// TwinCAT 3 PLC project Untitled1
// ProgramVersion: 3.1.4023.0
// libraries:
//   CmpBitmapPool, * (System)
//   Tc2_MC2, * (Beckhoff Automation GmbH)
//   Tc2_Standard, * (Beckhoff Automation GmbH)
//   Tc2_System, * (Beckhoff Automation GmbH)
//   Tc2_Utilities, * (Beckhoff Automation GmbH)
//   Tc3_Module, * (Beckhoff Automation GmbH)
//   Tc3_PackML_V2, * (Beckhoff Automation GmbH)
// project tree:
//   DUTs/ A21ToolStorage.TcDUT (not stored), Bundle.TcDUT (not stored), EOAT.TcDUT (not stored), Interval.TcDUT (not stored), PositionMaterials.TcDUT (not stored)
//   DUTs/Enums/ A21.TcDUT (not stored), Chipboard.TcDUT (not stored), Homing.TcDUT (not stored), SectionEnum.TcDUT (not stored), Surface.TcDUT, WoodBunk.TcDUT (not stored)
//   DUTs/Insertion/Drives/ AirPiston.TcPOU (not stored), ClearLinkMC.TcPOU (not stored), SimplePiston.TcPOU (not stored)
//   DUTs/Insertion/ Insertion.TcPOU (not stored), SuctionPad.TcDUT (not stored)
//   DUTs/Insertion/Prototypes/ FBA_Drive.TcPOU (not stored), I_ContinuousDrive.TcIO (not stored), I_Drive.TcIO, I_PositionalDrive.TcIO (not stored), I_EncodedDrive.TcIO (not stored)
//   DUTs/Machines/ Conveyor.TcPOU, ConveyorMode.TcDUT (not stored), KukaRobot.TcPOU (not stored), RobotA21.TcPOU (not stored), StrapMachine.TcPOU (not stored)
//   DUTs/Material Holders/ MaterialHolder.TcPOU (not stored), MaterialSlot.TcDUT (not stored), SkidMagazine.TcPOU (not stored), StagingTable.TcPOU (not stored)
//   GVLs/ ContainerArrays.TcGVL (not stored), GVL.TcGVL (not stored), Hardware.TcGVL (not stored), Misc.TcGVL (not stored)
//   / PlcTask.TcTTO (not stored)
//   POUs/A21a - Chipboard/AOIs/ AOI_LoadChipboard.TcPOU (not stored)
//   POUs/A21b - Wood Bunk/AOIs/ AOI_LoadWoodBunk.TcPOU (not stored), AOI_WoodBunkAlarms.TcPOU (not stored), AOI_StageWoodBunk.TcPOU (not stored), AOI_StagingTemplate.TcPOU (not stored)
//   POUs/ FB_System.TcPOU (not stored), MAIN.TcPOU
//   POUs/Hardware Calls/ InsertionQuality.TcPOU (not stored), SetSuctionsPtrArr.TcPOU (not stored), SuctionQuality.TcPOU (not stored), CallHardware.TcPOU (not stored), SetSuctions.TcPOU (not stored), SetupHardware.TcPOU (not stored)
//   POUs/A21a - Chipboard/ ChipboardEx.TcPOU (not stored)
//   POUs/A21b - Wood Bunk/ WoodBunkEx.TcPOU
//   POUs/Utility/ AddToStringArray.TcPOU (not stored), ArrayIsEmpty.TcPOU (not stored), BoolVLArrayToInteger.TcPOU (not stored), BoolPtrArrayToInteger.TcPOU (not stored), CleanStringsArray.TcPOU (not stored), IntegerBitAccess.TcPOU (not stored), IntegerToBoolArray.TcPOU (not stored), JoinStrings.TcPOU (not stored), WithinTolerance.TcPOU (not stored)

// ---- DUTs/Enums/Surface.TcDUT
{attribute 'qualified_only'}
{attribute 'strict'}
TYPE Surface :
(
	NULL,
	
	TOP,
	LEFT,
	RIGHT,
	BOTTOM,
	TOP_LEFT,
	TOP_RIGHT,
	BOTTOM_LEFT,
	BOTTOM_RIGHT,
	
	size
);
END_TYPE

// ---- DUTs/Insertion/Prototypes/I_Drive.TcIO
INTERFACE I_Drive

{attribute 'monitoring':='call'}
PROPERTY ABSTRACT AtHome : BOOL
GET
END_GET
END_PROPERTY

{attribute 'monitoring':='call'}
PROPERTY ABSTRACT AtInnerLimit : BOOL
GET
END_GET
END_PROPERTY

{attribute 'monitoring':='call'}
PROPERTY ABSTRACT AtOuterLimit : BOOL
GET
END_GET
END_PROPERTY

{attribute 'monitoring':='call'}
PROPERTY ABSTRACT Busy : BOOL
GET
END_GET
END_PROPERTY

{attribute 'monitoring':='call'}
PROPERTY ABSTRACT Contact : BOOL
GET
END_GET
END_PROPERTY

{attribute 'monitoring':='call'}
PROPERTY ABSTRACT Error : BOOL
GET
END_GET
END_PROPERTY

{attribute 'monitoring':='call'}
PROPERTY ABSTRACT HomeSet : BOOL
GET
END_GET
END_PROPERTY

METHOD ABSTRACT homingSequence : BOOL
VAR_INPUT
END_VAR
END_METHOD

METHOD reset : BOOL
VAR_INPUT
END_VAR
END_METHOD

METHOD ABSTRACT stop : BOOL
VAR_INPUT
END_VAR
END_METHOD

END_INTERFACE

// ---- DUTs/Machines/Conveyor.TcPOU
FUNCTION_BLOCK Conveyor
VAR_OUTPUT
	operation : ConveyorMode;
	request : ConveyorMode;
	
	enable AT %Q* : BOOL := TRUE;
	direction AT %Q* : BOOL; //FALSE = forward, TRUE = backward
	pulse AT %Q* : BOOL;
	reset AT %Q* : BOOL;
	
	error AT %I* : BOOL;
	sensorEntry AT %I* : BOOL;
	sensorExit AT %I* : BOOL;
	
	//vertical conveyors only
	requestLifter: BOOL;

	lifterEnable AT %Q* : BOOL := TRUE;
	lifterDirection AT %Q* : BOOL; //FALSE = up, TRUE = down
	lifterPulse AT %Q* : BOOL;
	lifterReset AT %Q* : BOOL;
	
	lifterError AT %I* : BOOL;
	extended AT %I* : BOOL;
	retracted AT %I* : BOOL;
END_VAR
VAR_OUTPUT
	position AT %I* : REAL;
	velocity AT %I* : REAL;
END_VAR
VAR
	hasLifter : BOOL;
	lifterMode : (HOLD, UP, DOWN);
	
	//pulses are assumed to be low-high-low
	pulser : TP;
	lifterPulser : TP;
	
END_VAR
VAR_STAT CONSTANT
	pulseWidth : TIME := T#25MS;
END_VAR

//conveyors do not move independently like motion drives, their operation is set by an additional conveyor control module
traverseSequence();
	
lifterPulser(IN:= , PT:= pulseWidth, Q=> lifterPulse, ET=> );
lifterPulser.IN := 
	hasLifter AND
	lifterEnable AND 
	NOT lifterError AND 
	NOT lifterReset AND 
	requestLifter AND
	lifterPulser.Q; //ends pulse itself

IF
	(extended AND lifterMode = UP) OR
	(retracted AND lifterMode = DOWN)
THEN
	lifterMode := HOLD;
END_IF

CASE lifterMode OF
	HOLD:
		lifterDirection := TRUE;
		lifterPulse := FALSE;
		
	UP:
		lifterDirection := FALSE;
		lifterPulse := NOT lifterPulse;
	
	DOWN:
		lifterDirection := TRUE;
		lifterPulse := NOT lifterPulse;
	
	
END_CASE

METHOD backward : BOOL
VAR_INPUT
END_VAR
END_METHOD

METHOD extend : BOOL
VAR_INPUT
END_VAR
VAR
	noLifter : BOOL;
END_VAR
IF hasLifter THEN
	lifterMode := UP;
	extend := TRUE;
ELSE
	noLifter := TRUE;
END_IF
END_METHOD

METHOD forward : BOOL
VAR_INPUT
END_VAR
END_METHOD

METHOD occupied : BOOL
occupied := sensorExit OR sensorEntry;
END_METHOD

METHOD reset : BOOL
VAR_INPUT
END_VAR
position := 0;
velocity := velocity; //no change

extend();
END_METHOD

METHOD retract : BOOL
VAR_INPUT
END_VAR
VAR
	noLifter : BOOL;
END_VAR
IF hasLifter THEN
	lifterMode := DOWN;
	retract := TRUE;
ELSE
	noLifter := TRUE;
END_IF
END_METHOD

METHOD setOperation : BOOL
VAR_INPUT
	newOperation : ConveyorMode;
END_VAR
operation := newOperation;
END_METHOD

METHOD setRequest : BOOL
VAR_INPUT
	requestedMode : ConveyorMode;
END_VAR
request := requestedMode;
END_METHOD

METHOD target : BOOL
VAR_INPUT
	targetPosition : REAL;
END_VAR
END_METHOD

METHOD PRIVATE traverseSequence : BOOL
VAR_INPUT
END_VAR
direction := (operation = ConveyorMode.BACKWARD);

pulser(IN:= , PT:= pulseWidth, Q=> pulse, ET=> );
pulser.IN := 
	enable AND 
	NOT error AND 
	NOT reset AND 
	(operation = ConveyorMode.FORWARD OR operation = ConveyorMode.BACKWARD)
	AND pulser.Q; //ends pulse itself
END_METHOD

END_FUNCTION_BLOCK

// ---- POUs/MAIN.TcPOU
PROGRAM MAIN
VAR
	stop : BOOL;
	manualStep : BOOL := TRUE;
	manualSuction : BOOL;
	
	moduleWB : WoodBunkEx;
	moduleCIP : ChipboardEx;
	
	exec1 : BOOL;
	exec2 : BOOL;
END_VAR

CallHardware(); //start program with hardware call - pass values and arrays into function blocks
SetupHardware(); //initialize values

runModules(); //LLD

CallHardware(); //end program with hardware call

ACTION runModules:
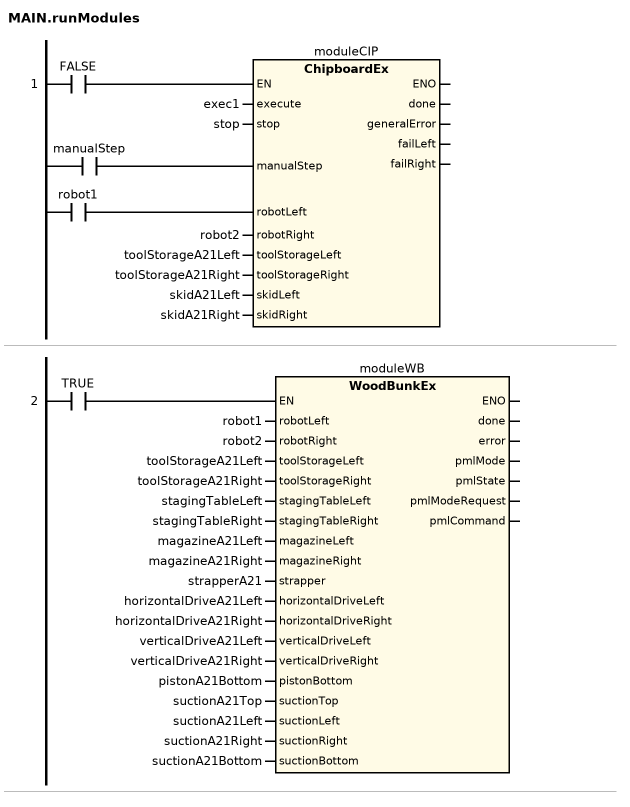
// NETWORK 1
IF FALSE THEN
    moduleCIP(
        execute := exec1,
        stop := stop,
        manualStep := manualStep,
        robotLeft := robot1,
        robotRight := robot2,
        toolStorageLeft := toolStorageA21Left,
        toolStorageRight := toolStorageA21Right,
        skidLeft := skidA21Left,
        skidRight := skidA21Right); // ChipboardEx
END_IF

// NETWORK 2
moduleWB(
    robotLeft := robot1,
    robotRight := robot2,
    toolStorageLeft := toolStorageA21Left,
    toolStorageRight := toolStorageA21Right,
    stagingTableLeft := stagingTableLeft,
    stagingTableRight := stagingTableRight,
    magazineLeft := magazineA21Left,
    magazineRight := magazineA21Right,
    strapper := strapperA21,
    horizontalDriveLeft := horizontalDriveA21Left,
    horizontalDriveRight := horizontalDriveA21Right,
    verticalDriveLeft := verticalDriveA21Left,
    verticalDriveRight := verticalDriveA21Right,
    pistonBottom := pistonA21Bottom,
    suctionTop := suctionA21Top,
    suctionLeft := suctionA21Left,
    suctionRight := suctionA21Right,
    suctionBottom := suctionA21Bottom); // WoodBunkEx
END_ACTION

END_PROGRAM

// ---- POUs/A21b - Wood Bunk/WoodBunkEx.TcPOU
FUNCTION_BLOCK WoodBunkEx
VAR_IN_OUT //references to required hardware
	robotLeft, robotRight : RobotA21;
	toolStorageLeft, toolStorageRight : A21ToolStorage;
	
	stagingTableLeft, stagingTableRight : StagingTable;
	magazineLeft, magazineRight : SkidMagazine;
	
	strapper : StrapMachine;
	
	horizontalDriveLeft, horizontalDriveRight : AirPiston;
	verticalDriveLeft, verticalDriveRight : ClearLinkMC;
	pistonBottom : SimplePiston;
	
	suctionTop : ARRAY[*] OF SuctionPad; (*1..3*)
	suctionLeft : ARRAY[*] OF SuctionPad; (*1..4*)
	suctionRight : ARRAY[*] OF SuctionPad; (*1..4*)
	suctionBottom : ARRAY[*] OF SuctionPad; (*1..2*)
END_VAR
VAR //controls
	stop : BOOL;
	execute : BOOL;
	hold : BOOL;
	reset : BOOL;
END_VAR
VAR_OUTPUT
	done : BOOL;
	error : BOOL;
	
	pmlMode : E_PMLProtectedUnitMode;
	pmlState : E_PMLState;
	pmlModeRequest : E_PMLProtectedUnitMode := ePMLProtUnitMode_Production;
	pmlCommand : E_PMLCommand;
END_VAR
VAR
	pmlModeString : STRING;
	pmlStateString : STRING;
	
	pmlStateMachine : PML_StateMachine;
	pmlModeManager : PML_UnitModeManager;

	step : (IDLE, STAGING, LOAD_WB, PUSH, STRAP, RELEASE, COMPLETE := 1050);
	iPair : INT;
	
	stageStepLeft, stageStepRight : INT;
	loadStepLeft, loadStepRight : INT;
END_VAR
VAR //local types
	insertionLeft, insertionRight : Insertion;
	
	demoHeight : REAL := 640; //mm
	materialsArr : ARRAY[0..GVL.maxPairs] OF PositionMaterials := [
		( position := 0, top := 'WDS20', left := 'WDS20', right := 'WDS20', bottom := 'WDB20' )];
		//( position := 69, top := 'WDS20', left := 'WDS20', right := 'WDS20', bottom := 'WDB20' )];
	
	loadedMaterials : ARRAY[Surface.TOP..Surface.BOTTOM] OF STRING;
END_VAR
VAR CONSTANT
	sectionID : SectionEnum := SectionEnum.WOOD_BUNK;
	suctionReleaseDelay : TIME := T#1000MS;
END_VAR
VAR
	//AOIs encapsulate functionality and reduce the number of module variables
	aoiTemplateLeft, aoiTemplateRight : AOI_StagingTemplate;
	aoiStageLeft, aoiStageRight : AOI_StageWoodBunk; 
	aoiLoadLeft, aoiLoadRight : AOI_LoadWoodBunk;
	
	suctionRelease : TON;
	
	//for testing, to be removed when deployoed
	latchLeft, latchRight : BOOL; //prevents SMC sliders from overshooting
	suctionEnableTop, suctionEnableLeft, suctionEnableRight, suctionEnableBottom : BOOL;
END_VAR

callLocalModules(); //initialize local modules

blocks(); //cyclically call AOIs and large library FBs

runPML(); //run PackML state machine

ACTION blocks:
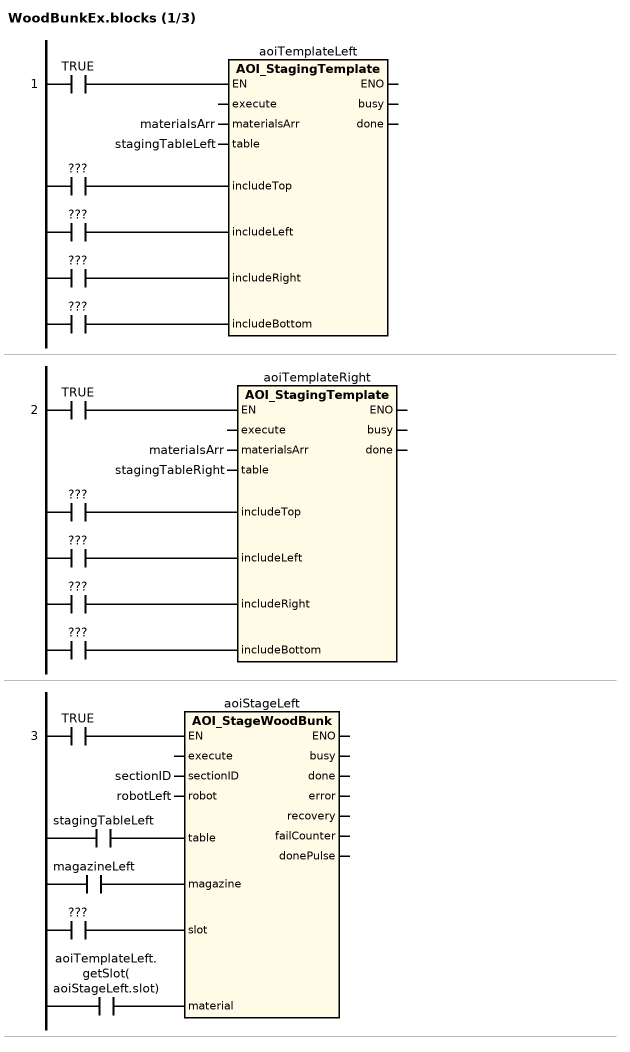
// NETWORK 1
aoiTemplateLeft(materialsArr := materialsArr, table := stagingTableLeft); // AOI_StagingTemplate

// NETWORK 2
aoiTemplateRight(materialsArr := materialsArr, table := stagingTableRight); // AOI_StagingTemplate

// NETWORK 3
aoiStageLeft(
    sectionID := sectionID,
    robot := robotLeft,
    table := stagingTableLeft,
    magazine := magazineLeft,
    material := aoiTemplateLeft.getSlot(aoiStageLeft.slot)); // AOI_StageWoodBunk

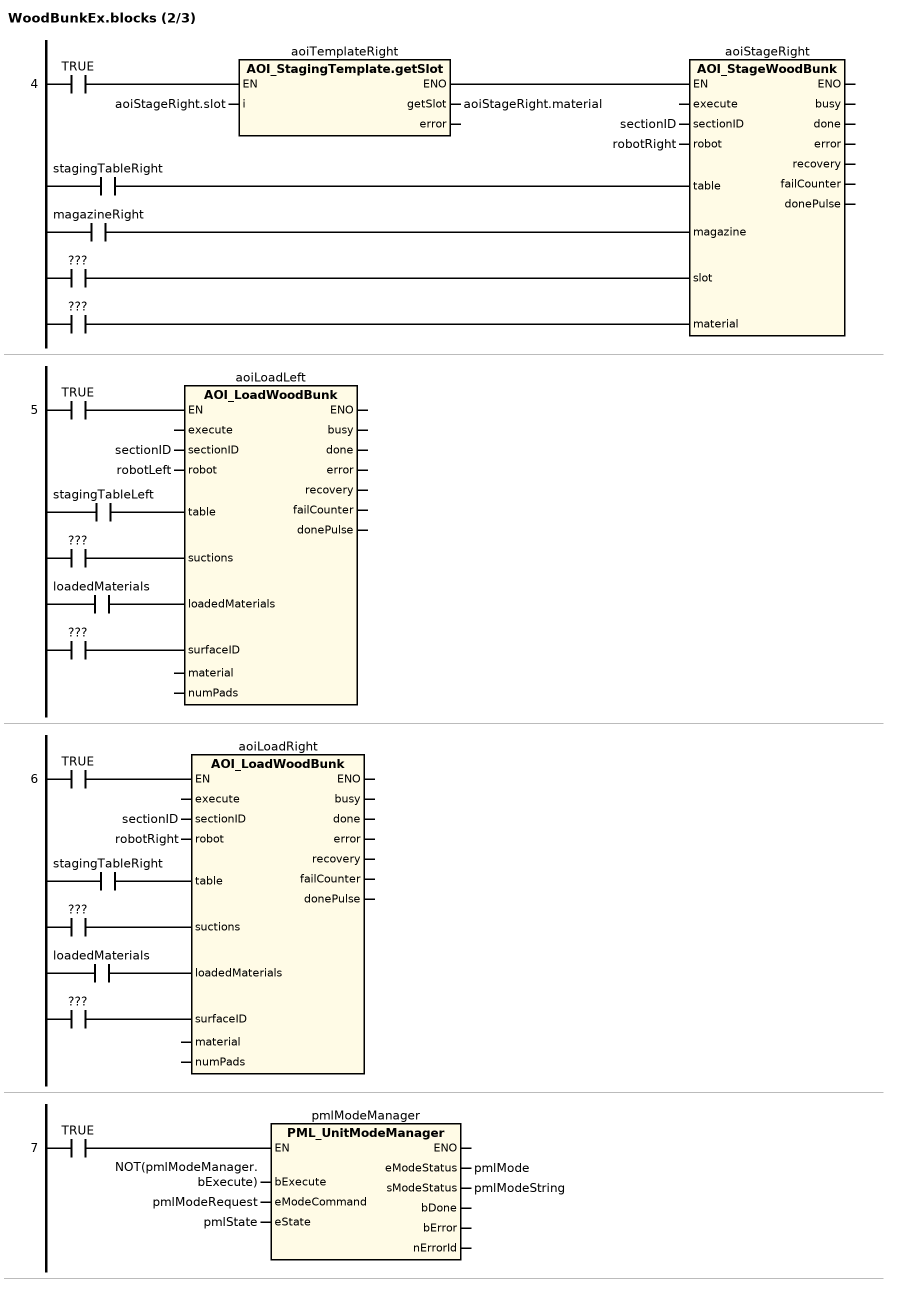
// NETWORK 4
aoiTemplateRight.getSlot(i := aoiStageRight.slot, getSlot => aoiStageRight.material);
aoiStageRight(
    sectionID := sectionID,
    robot := robotRight,
    table := stagingTableRight,
    magazine := magazineRight); // AOI_StageWoodBunk

// NETWORK 5
aoiLoadLeft(
    sectionID := sectionID,
    robot := robotLeft,
    table := stagingTableLeft,
    loadedMaterials := loadedMaterials); // AOI_LoadWoodBunk

// NETWORK 6
aoiLoadRight(
    sectionID := sectionID,
    robot := robotRight,
    table := stagingTableRight,
    loadedMaterials := loadedMaterials); // AOI_LoadWoodBunk

// NETWORK 7
pmlModeManager(
    bExecute := NOT(pmlModeManager.bExecute),
    eModeCommand := pmlModeRequest,
    eState := pmlState,
    eModeStatus => pmlMode,
    sModeStatus => pmlModeString); // PML_UnitModeManager

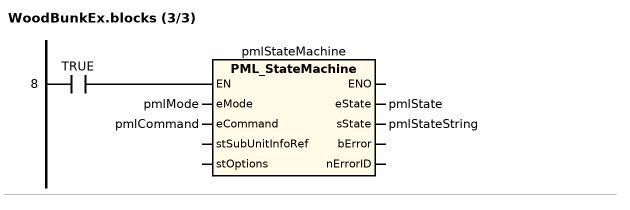
// NETWORK 8
pmlStateMachine(eMode := pmlMode, eCommand := pmlCommand, eState => pmlState, sState => pmlStateString); // PML_StateMachine
END_ACTION

ACTION callLocalModules:
{warning disable C0371}

insertionLeft(
	enable:= TRUE, 
	slider:= verticalDriveLeft, 
	screw:= horizontalDriveLeft, 
	contact=> , 
	softContact=> , 
	active=> , 
	error=> , 
	home=> , 
	homingComplete=> , 
	sliderPos=> );
	
insertionRight(
	enable:= TRUE, 
	slider:= verticalDriveRight, 
	screw:= horizontalDriveRight,  
	contact=> , 
	softContact=> , 
	active=> , 
	error=> , 
	home=> , 
	homingComplete=> , 
	sliderPos=> );
	
suctionRelease(IN:= , PT:= suctionReleaseDelay, Q=> , ET=> );
END_ACTION

METHOD PRIVATE load : BOOL
VAR_INPUT
	pairIndex : INT;
END_VAR
VAR_OUTPUT
	error : BOOL;
END_VAR
VAR
	pair : REFERENCE TO PositionMaterials REF= materialsArr[pairIndex];
	errorLeft, errorRight : BOOL;
END_VAR
{warning disable C0371}
(*
this is the new code for loading wood bunks from staging table to insertion
loading sequences are independent as each side has its own step variable
can be extended by changing the include<> parameters
*)

load :=
	loadEx(
		robot:= robotLeft, 
		aoiLoad:= aoiLoadLeft, 
		loadStep:= loadStepLeft, 
		pairIndex:= pairIndex, 
		includeTop:= TRUE, 
		includeLeft:= TRUE, 
		includeRight:= FALSE, 
		includeBottom:= FALSE, 
		error=> errorLeft)
	AND
	loadEx(
		robot:= robotRight, 
		aoiLoad:= aoiLoadRight, 
		loadStep:= loadStepRight, 
		pairIndex:= pairIndex, 
		includeTop:= FALSE, 
		includeLeft:= FALSE, 
		includeRight:= TRUE, 
		includeBottom:= TRUE, 
		error=> errorRight);
		
error := errorLeft OR errorRight;

(*
below is the old code for loading wood bunks from staging table to insertion
it loads wood bunks in sets - top/bottom, then sides
if one side is finished loading a set before the other, it waits until the other side is done before advancing the set
*)
(*
IF robotLeft.error OR robotRight.error THEN
	error := TRUE;
	RETURN;
	
ELSIF 
	(robotLeft.reservation <> sectionID AND_THEN NOT robotLeft.reserve(sectionID)) OR 
	(robotRight.reservation <> sectionID AND_THEN NOT robotRight.reserve(sectionID))
THEN //loading requires both robots be reserved together
	RETURN;
	
ELSIF //robots have wrong tool
	(robotLeft.tool <> sectionID AND_THEN NOT robotLeft.changeEOAT(targetTool := sectionID)) OR
	(robotRight.tool <> sectionID AND_THEN NOT robotRight.changeEOAT(targetTool := sectionID))
THEN
	RETURN;
	
END_IF

CASE loadStep OF
	0: //top and bottom
		IF aoiLoadLeft.done AND aoiLoadRight.done THEN
			aoiLoadLeft.execute := aoiLoadRight.execute := FALSE;
			aoiLoadLeft.material := aoiLoadRight.material := '';
			
			aoiLoadLeft.reset();
			aoiLoadRight.reset();
			loadStep := 10;
			RETURN;
		END_IF
		
		aoiLoadLeft.suctions := suctionTop;
		aoiLoadLeft.surfaceID := Surface.TOP;
		aoiLoadLeft.material := pair.top;
		aoiLoadLeft.numPads := UPPER_BOUND(suctionTop, 1) - LOWER_BOUND(suctionTop, 1) + 1;
		
		aoiLoadRight.suctions := suctionBottom;
		aoiLoadRight.surfaceID := Surface.BOTTOM;
		aoiLoadRight.material := pair.bottom;
		aoiLoadRight.numPads := UPPER_BOUND(suctionBottom, 1) - LOWER_BOUND(suctionBottom, 1) + 1;
		
		aoiLoadLeft.execute := NOT aoiLoadLeft.done AND NOT aoiLoadLeft.busy;
		aoiLoadRight.execute := NOT aoiLoadRight.done AND NOT aoiLoadRight.busy;
		
	10: //sides
		IF aoiLoadLeft.done AND aoiLoadRight.done THEN
			aoiLoadLeft.execute := aoiLoadRight.execute := FALSE;
			aoiLoadLeft.material := aoiLoadRight.material := '';
			
			aoiLoadLeft.reset();
			aoiLoadRight.reset();
			loadStep := COMPLETE;
			RETURN;
		END_IF
		
		aoiLoadLeft.suctions := suctionLeft;
		aoiLoadLeft.surfaceID := Surface.LEFT;
		aoiLoadLeft.material := pair.left;
		aoiLoadLeft.numPads := UPPER_BOUND(suctionLeft, 1) - LOWER_BOUND(suctionLeft, 1) + 1;
		
		aoiLoadRight.suctions := suctionRight;
		aoiLoadRight.surfaceID := Surface.RIGHT;
		aoiLoadRight.material := pair.right;
		aoiLoadRight.numPads := UPPER_BOUND(suctionRight, 1) - LOWER_BOUND(suctionRight, 1) + 1;
		
		aoiLoadLeft.execute := NOT aoiLoadLeft.done AND NOT aoiLoadLeft.busy;
		aoiLoadRight.execute := NOT aoiLoadRight.done AND NOT aoiLoadRight.busy;
		
	COMPLETE:				
		robotLeft.release(sectionID);
		robotRight.release(sectionID);
		
		aoiLoadLeft.material := aoiLoadRight.material := '';
		aoiLoadLeft.execute := aoiLoadRight.execute := FALSE;
		
		loadStep := 0;
		load := TRUE;
END_CASE

//--------------------------------------------------
IF aoiLoadLeft.recovery THEN //if loading in recovery mode - refill table, resume loading when finished
	aoiLoadLeft.execute := stageEx(
		robot:= robotLeft, 
		aoiTemplate:= aoiTemplateLeft, 
		aoiStaging:= aoiStageLeft, 
		stageStep:= stageStepLeft, 
		includeTop:= TRUE, 
		includeLeft:= TRUE, 
		includeRight:= FALSE, 
		includeBottom:= FALSE, 
		error=> );
ELSE
	//loadLeft.execute := NOT loadLeft.busy AND NOT loadLeft.done;
END_IF
//--------------------------------------------------
IF aoiLoadRight.recovery THEN
	aoiLoadRight.execute := stageEx(
		robot:= robotRight, 
		aoiTemplate:= aoiTemplateRight, 
		aoiStaging:= aoiStageRight, 
		stageStep:= stageStepRight, 
		includeTop:= FALSE, 
		includeLeft:= FALSE, 
		includeRight:= TRUE, 
		includeBottom:= TRUE, 
		error=> );
ELSE
	//loadRight.execute := NOT loadRight.busy AND NOT loadRight.done;
END_IF
//--------------------------------------------------
	
error := aoiLoadLeft.error OR aoiLoadRight.error;
*)
END_METHOD

METHOD PRIVATE loadEx : BOOL
VAR_IN_OUT
	robot : RobotA21;
	aoiLoad : AOI_LoadWoodBunk;
	loadStep : INT;
END_VAR
VAR_INPUT
	pairIndex : INT;
	includeTop, includeLeft, includeRight, includeBottom : BOOL;
END_VAR
VAR_OUTPUT
	error : BOOL;
END_VAR
VAR
	pair : REFERENCE TO PositionMaterials REF= materialsArr[pairIndex];
END_VAR
{warning disable C0371}
IF robot.error THEN
	error := TRUE;
	RETURN;
ELSIF robot.reservation <> sectionID AND_THEN NOT robot.reserve(sectionID) THEN
	RETURN;
ELSIF robot.tool <> sectionID AND_THEN NOT robot.changeEOAT(targetTool := sectionID) THEN
	RETURN;
END_IF

error := aoiLoad.error;

CASE loadStep OF
	0:
		loadStep := Surface.TOP;
	
	Surface.TOP:		
		IF NOT includeTop OR aoiLoad.donePulse THEN
			aoiLoad.execute := FALSE;
			aoiLoad.material := '';
			loadStep := Surface.BOTTOM;
			RETURN;
		END_IF
		
		aoiLoad.surfaceID := Surface.TOP;
		aoiLoad.material := pair.top;
		aoiLoad.suctions := suctionTop;
		aoiLoad.numPads := UPPER_BOUND(suctionTop, 1) - LOWER_BOUND(suctionTop, 1) + 1;
		
		aoiLoad.execute := NOT aoiLoad.busy;
		
	Surface.BOTTOM:
		IF NOT includeBottom OR aoiLoad.donePulse THEN
			aoiLoad.execute := FALSE;
			aoiLoad.material := '';
			loadStep := Surface.LEFT;
			RETURN;
		END_IF
		
		aoiLoad.surfaceID := Surface.BOTTOM;
		aoiLoad.material := pair.bottom;
		aoiLoad.suctions := suctionBottom;
		aoiLoad.numPads := UPPER_BOUND(suctionBottom, 1) - LOWER_BOUND(suctionBottom, 1) + 1;
		
		aoiLoad.execute := NOT aoiLoad.busy;
		
	Surface.LEFT:
		IF NOT includeLeft OR aoiLoad.donePulse THEN
			aoiLoad.execute := FALSE;
			aoiLoad.material := '';
			loadStep := Surface.RIGHT;
			RETURN;
		END_IF
		
		aoiLoad.surfaceID := Surface.LEFT;
		aoiLoad.material := pair.left;
		aoiLoad.suctions := suctionLeft;
		aoiLoad.numPads := UPPER_BOUND(suctionLeft, 1) - LOWER_BOUND(suctionLeft, 1) + 1;
		
		aoiLoad.execute := NOT aoiLoad.busy;
		
	Surface.RIGHT:
		IF NOT includeRight OR aoiLoad.donePulse THEN
			aoiLoad.execute := FALSE;
			aoiLoad.material := '';
			loadStep := COMPLETE;
			RETURN;
		END_IF
		
		aoiLoad.surfaceID := Surface.RIGHT;
		aoiLoad.material := pair.right;
		aoiLoad.suctions := suctionRight;
		aoiLoad.numPads := UPPER_BOUND(suctionRight, 1) - LOWER_BOUND(suctionRight, 1) + 1;
		
		aoiLoad.execute := NOT aoiLoad.busy;
		
	COMPLETE:				
		robot.release(sectionID);
		
		aoiLoad.material := '';
		aoiLoad.execute := FALSE;
		
		loadEx := TRUE;
END_CASE
END_METHOD

METHOD PRIVATE maintenance : BOOL
VAR_INPUT
END_VAR
{warning disable C0371}
//no specific tasks yet, free run and testing
SetSuctions(suctionTop, suctionEnableTop);
SetSuctions(suctionLeft, suctionEnableLeft);
SetSuctions(suctionRight, suctionEnableRight);
SetSuctions(suctionBottom, suctionEnableBottom);

IF robotLeft.Done THEN
	robotLeft.clearCommand();
END_IF

IF robotRight.Done THEN
	robotRight.clearCommand();
END_IF
END_METHOD

METHOD PRIVATE process : BOOL
VAR_INPUT
	manualMode : BOOL;
END_VAR
{warning disable C0371}
CASE step OF
	IDLE:
		step := STAGING;
		
	STAGING:
		IF NOT done THEN
			done := stage(); //calls stageEx() for both robots
		END_IF
		
		IF
			(manualMode AND_THEN execute) OR
			(NOT manualMode AND_THEN done)
		THEN
			robotLeft.clearCommand();
			robotRight.clearCommand();
			
			aoiStageLeft.reset();
			aoiStageRight.reset();
			
			stageStepLeft := stageStepRight := 0;
			
			execute := FALSE;
			done := FALSE;
			step := LOAD_WB;
		END_IF
	
	LOAD_WB:
		IF NOT done THEN
			done := load(pairIndex := iPair, error => error);
		END_IF
		
		IF manualMode THEN
			SetSuctions(suctionTop, suctionEnableTop);
			SetSuctions(suctionLeft, suctionEnableLeft);
			SetSuctions(suctionRight, suctionEnableRight);
			SetSuctions(suctionBottom, suctionEnableBottom);
		END_IF
		
		IF
			(manualMode AND_THEN execute) OR
			(NOT manualMode AND_THEN done)
		THEN
			robotLeft.clearCommand();
			robotRight.clearCommand();
			
			aoiLoadLeft.reset();
			aoiLoadRight.reset();
			
			loadStepLeft := loadStepRight := 0;
			stageStepLeft := stageStepRight := 0;
			
			done := FALSE;
			suctionEnableTop := suctionEnableLeft := suctionEnableRight := suctionEnableBottom := FALSE;
			execute := FALSE;
			
			step := PUSH;
		END_IF
		
	PUSH:
		IF
			(manualMode AND_THEN execute) OR
			(NOT manualMode AND latchLeft AND latchRight AND pistonBottom.extended)
		THEN
			insertionLeft.stop();
			insertionRight.stop();
			
			latchLeft := latchRight := FALSE;
			execute := FALSE;
			step := STRAP;
			RETURN;
		END_IF
		
		IF NOT validateInsertion(checkTop:= FALSE, checkLeft:= FALSE, checkRight:= FALSE, checkBottom:= FALSE) THEN
			error := TRUE;
			RETURN;
		END_IF
		(*
		IF 
			insertionLeft.sliderPos <> demoHeight/2 //OR 
			//insertionRight.sliderPos <> demoHeight/2 //OR 
			//NOT insertionBottom.contact
		THEN
			insertionLeft.slideAbsolute(demoHeight/2);
			//insertionRight.slideAbsolute(demoHeight/2);
			RETURN;
		END_IF
		*)
		
		IF insertionLeft.screw.Contact THEN
			latchLeft := TRUE;
		ELSIF NOT latchLeft THEN
			insertionLeft.press();
		END_IF
		
		IF insertionRight.screw.Contact THEN
			latchRight := TRUE;
		ELSIF NOT latchRight THEN
			insertionRight.press();
		END_IF
		pistonBottom.extend();
		
	STRAP:	
		strapper.bEnable := TRUE;
		IF strapper.done THEN
			suctionRelease.IN := FALSE;
			step := RELEASE;
			RETURN;
		END_IF
		
		IF suctionRelease.Q THEN
			SetSuctions(suctionTop, FALSE);
			SetSuctions(suctionLeft, FALSE);
			SetSuctions(suctionRight, FALSE);
			SetSuctions(suctionBottom, FALSE);
		ELSIF strapper.atBundleLevel THEN
			suctionRelease.IN := TRUE;
		END_IF
		
		IF strapper.ready THEN
			strapper.strap();
		END_IF
		
		IF execute THEN
			suctionRelease.IN := FALSE;
			execute := FALSE;
			step := RELEASE;
		END_IF
		
	RELEASE: //release command		
		//insertionLeft.slideAbsolute(0);
		//insertionRight.slideAbsolute(0);
		
		insertionLeft.release();
		insertionRight.release();
		pistonBottom.retract();
		
		IF 
			(insertionLeft.screw.AtHome AND insertionRight.screw.AtHome AND pistonBottom.retracted) OR
			execute
		THEN
			execute := FALSE;
			step := COMPLETE;
		END_IF
	
	COMPLETE:
		//reset everything
		iPair := (iPair + 1) MOD GVL.maxPairs;
		step := IDLE;
		
		process := TRUE;
END_CASE
END_METHOD

METHOD PRIVATE ps_Aborting : BOOL
VAR_INPUT
END_VAR
{warning disable C0371}
insertionLeft.stop();
insertionRight.stop();
pistonBottom.stop();

aoiLoadLeft.reset();
aoiLoadRight.reset();

aoiStageLeft.reset();
aoiStageRight.reset();

robotLeft.clearCommand();
robotRight.clearCommand();

//stop conveyors

ps_Aborting :=
	NOT insertionLeft.active AND
	NOT insertionRight.active AND
	NOT pistonBottom.busy AND
	NOT robotLeft.Busy AND
	NOT robotRight.Busy;
END_METHOD

METHOD PRIVATE ps_Clearing : BOOL
VAR_INPUT
END_VAR
{warning disable C0371}
insertionLeft.reset();
insertionRight.reset();

ps_Clearing := 
	NOT insertionLeft.error AND
	NOT insertionRight.error AND
	NOT strapper.error AND
	NOT robotLeft.error AND
	NOT robotRight.error;
END_METHOD

METHOD PRIVATE ps_Execute : BOOL
VAR_INPUT
END_VAR
CASE pmlMode OF
	0: //invalid mode
	ePMLProtUnitMode_Production:	ps_Execute := process(manualMode := FALSE);
	ePMLProtUnitMode_Maintenance:	maintenance();
	ePMLProtUnitMode_Manual:		ps_Execute := process(manualMode := TRUE);
END_CASE
END_METHOD

METHOD PRIVATE ps_Holding : BOOL
VAR_INPUT
END_VAR
{warning disable C0371}
insertionLeft.stop();
insertionRight.stop();
pistonBottom.stop();
//set robot to pause
pmlStateMachine.M_StateComplete();
END_METHOD

METHOD PRIVATE ps_Resetting : BOOL
VAR_INPUT
END_VAR
{warning disable C0371}
insertionLeft.reset();
insertionRight.reset();

ps_Resetting := 
	reset AND
	NOT insertionLeft.error AND
	NOT insertionRight.error AND
	NOT strapper.error AND
	NOT robotLeft.error AND
	NOT robotRight.error;
END_METHOD

METHOD PRIVATE ps_Stopping : BOOL
VAR_INPUT
END_VAR
{warning disable C0371}
insertionLeft.stop();
insertionRight.stop();
pistonBottom.stop();

aoiLoadLeft.reset();
aoiLoadRight.reset();

aoiStageLeft.reset();
aoiStageRight.reset();

robotLeft.clearCommand();
robotRight.clearCommand();

//stop conveyors

ps_Stopping :=
	NOT insertionLeft.active AND
	NOT insertionRight.active AND
	NOT pistonBottom.busy AND
	NOT robotLeft.Busy AND
	NOT robotRight.Busy;
END_METHOD

ACTION runPML:
(*
PackML
	state machine for packaging applications - see Tc3_PackML_V2 library on InfoSys
	
	final states - wait for an input or condition and command to new state
	intermediate states - complete a task and call pmlStateMachine.M_StateComplete() to advance to next state
	
the following states currently use the same logic (albeit in different methods), implementation may change later
	ps_Stopping() and ps_Aborting()
	ps_Resetting() and ps_Clearing()
	
STOP - controlled stop **with intent to shutdown or vacate for extended time** induced by operator/HMI - otherwise use HOLD
ABORT - emergency stop due to machine errors


HOLD - minor local issues
SUSPEND - external issues

EXECUTE - major control logic
	different modes may require different tasks
	create methods as required for different modes, then call the correct method in ps_Completing()
	can be commanded to STOP, ABORT, HOLD, or SUSPEND at any point
COMPLETING - process complete, move product out of system and finish transition to COMPLETED
*)

IF //abort at machine error
	insertionLeft.error OR 
	insertionRight.error OR 
	robotLeft.error OR 
	robotRight.error OR
	strapper.error
THEN
	pmlCommand := ePMLCommand_Abort;
	
ELSIF stop THEN //stop at command stop
	pmlCommand := ePMLCommand_Stop;

ELSIF FALSE (*A2.4 cannot allow bundles to enter*) THEN //FALSE condition never executes - this is temporary
	pmlCommand := ePMLCommand_Suspend;
END_IF


CASE pmlState OF
	0: (*ePMLState_Undefined*) //default state on startup
		pmlCommand := ePMLCommand_Stop;
		
	ePMLState_Stopping:
		IF ps_Stopping() THEN
			pmlStateMachine.M_StateComplete();
		END_IF
		
	ePMLState_Stopped:
		pmlCommand := ePMLCommand_Reset;
	
    ePMLState_Resetting:
		IF ps_Resetting() THEN
			reset := FALSE;
			pmlStateMachine.M_StateComplete();
		END_IF
		
	ePMLState_Idle:
		IF execute THEN
			execute := FALSE;
			//suctionEnableTop := suctionEnableLeft := suctionEnableRight := suctionEnableBottom := FALSE;
			pmlCommand := ePMLCommand_Start;
		END_IF		
		(*
		SetSuctions(suctionTop, suctionEnableTop);
		SetSuctions(suctionLeft, suctionEnableLeft);
		SetSuctions(suctionRight, suctionEnableRight);
		SetSuctions(suctionBottom, suctionEnableBottom);
		*)
	
	ePMLState_Starting:
		IF insertionLeft.screw.HomeSet AND insertionRight.screw.HomeSet AND pistonBottom.retracted THEN
			pmlStateMachine.M_StateComplete();
			
		ELSE //homing sequence
			robotLeft.clearCommand();
			robotRight.clearCommand();
			
			insertionLeft.homingSequence();
			insertionRight.homingSequence();
			pistonBottom.retract();
		END_IF
	
	ePMLState_Execute: 
		IF hold THEN
			pmlCommand := ePMLCommand_Hold;
		END_IF
		IF ps_Execute() THEN
			pmlStateMachine.M_StateComplete();
			pmlCommand := ePMLCommand_Complete;
		END_IF
		
	ePMLState_Completing:
		pmlStateMachine.M_StateComplete();
	
	ePMLState_Complete:
		pmlCommand := ePMLCommand_Reset;
	
	ePMLState_Holding:
		IF ps_Holding() THEN
			pmlStateMachine.M_StateComplete();
		END_IF
	
	ePMLState_Held:
		IF NOT hold THEN
			pmlCommand := ePMLCommand_Unhold;
		END_IF
	
	ePMLState_Unholding:
		pmlStateMachine.M_StateComplete(); //release all pause commands and IO
	
	ePMLState_Suspended: //based on output section conditions
	ePMLState_Suspending: //based on output section conditions
	ePMLState_Unsuspending: //based on output section conditions
	
	ePMLState_Aborting:
		IF ps_Aborting() THEN
			pmlStateMachine.M_StateComplete();
		END_IF
	
	ePMLState_Aborted:
		pmlCommand := ePMLCommand_Clear;
	
	ePMLState_Clearing:
		IF ps_Clearing() THEN
			pmlStateMachine.M_StateComplete();
		END_IF
	
END_CASE
END_ACTION

METHOD PRIVATE stage : BOOL
VAR_OUTPUT
	error : BOOL;
END_VAR
{warning disable C0371}

(*
this method only exists to call stageEx() for both robots
*)
(*
stage := leftDone AND rightDone;

IF NOT leftDone THEN
	leftDone := stageEx(
		robot:= robotLeft, 
		aoiTemplate:= aoiTemplateLeft, 
		aoiStaging:= aoiStageLeft, 
		stageStep:= stageStepLeft, 
		//iSlot:= iSlotLeft, 
		includeTop:= TRUE, 
		includeLeft:= TRUE, 
		includeRight:= FALSE, 
		includeBottom:= FALSE, 
		error=> );
END_IF

IF NOT rightDone THEN
	rightDone := stageEx(
		robot:= robotRight, 
		aoiTemplate:= aoiTemplateRight, 
		aoiStaging:= aoiStageRight, 
		stageStep:= stageStepRight, 
		//iSlot:= iSlotRight, 
		includeTop:= FALSE, 
		includeLeft:= FALSE, 
		includeRight:= TRUE, 
		includeBottom:= TRUE, 
		error=> );
END_IF
*)

stage := 
	stageEx(
		robot:= robotLeft, 
		aoiTemplate:= aoiTemplateLeft, 
		aoiStaging:= aoiStageLeft, 
		stageStep:= stageStepLeft, 
		includeTop:= TRUE, 
		includeLeft:= TRUE, 
		includeRight:= FALSE, 
		includeBottom:= FALSE, 
		error=> )
	AND
	stageEx(
		robot:= robotRight, 
		aoiTemplate:= aoiTemplateRight, 
		aoiStaging:= aoiStageRight, 
		stageStep:= stageStepRight, 
		includeTop:= FALSE, 
		includeLeft:= FALSE, 
		includeRight:= TRUE, 
		includeBottom:= TRUE, 
		error=> );
END_METHOD

METHOD PRIVATE stageEx : BOOL
VAR_IN_OUT
	robot : RobotA21;
	aoiTemplate : AOI_StagingTemplate;
	aoiStaging : AOI_StageWoodBunk;
	stageStep : INT;
END_VAR
VAR_INPUT
	includeTop, includeLeft, includeRight, includeBottom : BOOL;
END_VAR
VAR_OUTPUT
	error : BOOL;
END_VAR
{warning disable C0371}
IF robot.error THEN
	error := TRUE;
	RETURN;
ELSIF robot.reservation <> sectionID AND_THEN NOT robot.reserve(sectionID) THEN
	RETURN;
ELSIF robot.tool <> sectionID AND_THEN NOT robot.changeEOAT(targetTool := sectionID) THEN
	RETURN;
END_IF

CASE stageStep OF
	0: //generate staging template
		IF aoiTemplate.done THEN
			aoiTemplate.execute := FALSE;
			stageStep := 10;
			RETURN;
		END_IF
		
		aoiTemplate.execute := NOT aoiTemplate.busy;
		
		aoiTemplate.includeTop := includeTop;
		aoiTemplate.includeLeft := includeLeft;
		aoiTemplate.includeRight := includeRight;
		aoiTemplate.includeBottom := includeBottom;
		
	10: //stage tables
		IF aoiStaging.slot > 10 THEN
			aoiStaging.execute := FALSE;			
			stageStep := COMPLETE;
			RETURN;
		END_IF
		
		aoiStaging.execute := NOT aoiStaging.busy; //execute if aoiStaging is ready
		
		aoiStaging.slot := MAX(1, aoiStaging.slot); //if 0, sets to 1
		aoiStaging.slot := MIN(aoiStaging.slot, 999); //prevents overflow 
		
		IF aoiStaging.donePulse THEN
			aoiStaging.slot := aoiStaging.slot + 1;
		END_IF
	
	COMPLETE:
		aoiTemplate.clearTemplate();
		aoiTemplate.execute := FALSE;
		aoiStaging.execute := FALSE;
		aoiStaging.reset();
		
		robot.release(sectionID);
		
		aoiStaging.slot := 0;
		
		stageEx := TRUE;
		//stageStep := 0;
END_CASE

error := aoiStaging.error;
END_METHOD

METHOD PRIVATE validateInsertion : BOOL
VAR_INPUT
	checkTop : BOOL;
	checkLeft : BOOL;
	checkRight : BOOL;
	checkBottom : BOOL;
END_VAR
validateInsertion := 
	(NOT checkTop OR_ELSE SuctionQuality(suctions:= suctionTop)) AND
	(NOT checkLeft OR_ELSE SuctionQuality(suctions:= suctionLeft)) AND
	(NOT checkRight OR_ELSE SuctionQuality(suctions:= suctionRight)) AND
	(NOT checkBottom OR_ELSE SuctionQuality(suctions:= suctionBottom));

(*
validateSuctionQuality := 
	(
		NOT checkTop OR_ELSE InsertionQuality(
			suctions:= suctionTop, 
			insertionMaterial:= loadedMaterials[Surface.TOP], 
			recipeMaterial:= materialsArr[iPair].top)
	) AND
	(
		NOT checkLeft OR_ELSE InsertionQuality(
			suctions:= suctionLeft, 
			insertionMaterial:= loadedMaterials[Surface.LEFT], 
			recipeMaterial:= materialsArr[iPair].left)
	) AND
	(
		NOT checkRight OR_ELSE InsertionQuality(
			suctions:= suctionRight, 
			insertionMaterial:= loadedMaterials[Surface.RIGHT], 
			recipeMaterial:= materialsArr[iPair].right)
	) AND
	(
		NOT checkBottom OR_ELSE InsertionQuality(
			suctions:= suctionBottom, 
			insertionMaterial:= loadedMaterials[Surface.BOTTOM], 
			recipeMaterial:= materialsArr[iPair].bottom)
	);
*)
END_METHOD

END_FUNCTION_BLOCK
